FUNCTION_BLOCK OrderRegisterAgentFB (* Registers orders *)
  (* Standard: 61499-1 *)
  (* Version 1.0, 20010-04-20, AnLo, TUT *)
  (* Compiler header: package fb.rt; *)
  (* Compiler Java Sun JDK 1.5.0 *)
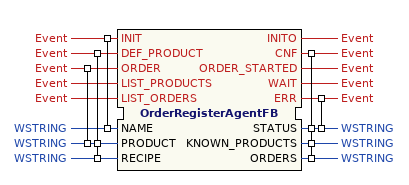
  EVENT_INPUT
    INIT WITH NAME; (* Initialization *)
    DEF_PRODUCT WITH PRODUCT, RECIPE; (* Define product *)
    ORDER WITH PRODUCT;
    LIST_PRODUCTS;
    LIST_ORDERS; (* List current orders *)
  END_EVENT
  EVENT_OUTPUT
    INITO; (* Block initialized *)
    CNF WITH STATUS, KNOWN_PRODUCTS, ORDERS; (* Confirmation event *)
    ORDER_STARTED;
    WAIT; (* Order cannot be intput now *)
    ERR WITH STATUS; (* Error while executing the request (E.g. unknown Product ordered: "PRODUCT_UNKNOWN. *)
  END_EVENT
  VAR_INPUT
    NAME : WSTRING; (* Input event qualifier *)
    PRODUCT : WSTRING;
    RECIPE : WSTRING;
  END_VAR
  VAR_OUTPUT
    STATUS : WSTRING;
    KNOWN_PRODUCTS : WSTRING;
    ORDERS : WSTRING; (* Lists # of orders: "{(A, 1), (B,2)}; {(A, 6), (B,7)}" = "Current Orders; Finalized Orders" *)
  END_VAR
END_FUNCTION_BLOCK
